INTERFACE ITcoKeyMode

PROPERTY KeyInAuto : BOOL
GET
END_GET
END_PROPERTY

PROPERTY KeyInManual : BOOL
GET
END_GET
END_PROPERTY

PROPERTY KeyInStep : BOOL
GET
END_GET
END_PROPERTY

END_INTERFACE

(* stored: Version 1.1.0.1
   Itf ITcoKeyMode: Id {2b49ab04-04e7-41a1-8dcf-5c197e466512}
   Property KeyInAuto: Id {fa94d403-8925-424a-8063-e48566c23b37}
   Get Get: Id {788e2838-1d2b-4f56-9330-21ba66c8e7c5}
   Property KeyInManual: Id {38cbc47b-948a-4b37-8a4c-a14c7eda2e32}
   Get Get: Id {93b02fa6-7dcb-4cb5-abb6-25f6d572dde9}
   Property KeyInStep: Id {39dcaa54-a72c-490b-b20f-8d061ddf3d6b}
   Get Get: Id {26792d85-6f80-473b-a5c7-7e8a5da8208d} *)
